# EPICS autosave request: ADmar345/mar345App/Db/mar345_settings.req
file "ADBase_settings.req", P=$(P), R=$(R)
file "NDFile_settings.req", P=$(P), R=$(R)
$(P)$(R)EraseMode
$(P)$(R)NumErase
$(P)$(R)ScanSize
$(P)$(R)ScanResolution
